TYPE ST_ManualModeState :
STRUCT
	arrAxisInG201: ARRAY[0..HLI_KEY_MAXIDX] OF UINT;
END_STRUCT
END_TYPE

(* stored: Version 1.1.0.1, ProductVersion 3.1.4019.0
   DUT ST_ManualModeState: Id {d19f6a8c-41ce-4eed-8591-94903df7e284} *)
